// TIA Portal V19 export
TYPE "LEXCHANGETRAY_typeConstraintRollerTranserfCondition"
// stored: Access Published
   STRUCT
      axisPosMoveCondition : Bool;
   END_STRUCT;
END_TYPE
